// TIA Portal V16 export
// export: Created 2021-04-06T19:52:19.1197079Z, ExportSetting WithDefaults, DisplayName Totally Integrated Automation Portal, DisplayVersion V16, DisplayName TIA Portal Version Control Interface, DisplayVersion V16, DisplayName TIA Portal Openness, DisplayVersion V16, DisplayName STEP 7 Professional, DisplayVersion V16, DisplayName STEP 7 Safety, DisplayVersion V16, DisplayName WinCC Unified SCADA Engineering System, DisplayVersion V16
TYPE "dataStantion"
// stored: IsFailsafeCompliant false
   STRUCT
      numberDozInMin : Int;   // число доз в минуту
      numberDozInthisWeight : Int;   // полученное число доз заданной порции
      nuvberDozSmena : Int;   // число доз за смену
      currentPogreshn1 : Real;   // погрешность для текущей дозы 1 машины
      currentPogr2 : Real;   // погрешность для текущей дозы 2 машины
      maxPogr : Real;   // максимальная погрешность для порции
      isEmulation : Bool;
      emulStartDozing : Array[0..2] of Bool;
      emulReadyAccept : Array[0..2] of Bool;
   END_STRUCT;
END_TYPE
